FUNCTION "LGF_MatrixSubtraction" : Void
TITLE = LGF_MatrixSubtraction
{ S7_Optimized_Access := 'TRUE' }
AUTHOR : Siemens_Digital_Industries
FAMILY : LGF
NAME : LGF_MatrixSubtraction
//This function subtracts a matrix of the data type `ARRAY[*,*] of LREAL` from another one.
//
//The individual fields of the two matrices are read, subtracted and then output in the matrix `matrixResult`.
//
//$$
// result =
//
//\begin{bmatrix}
//   a_{11} & \cdots & a_{1n} \\
//   \vdots & \ddots & \vdots \\
//   a_{m1} & \cdots & a_{mn}
//\end{bmatrix}
//
//-
//
//\begin{bmatrix}
//   b_{11} & \cdots & b_{1n} \\
//   \vdots & \ddots & \vdots \\
//   b_{m1} & \cdots & b_{mn}
//\end{bmatrix}
//
//=
//
//\begin{bmatrix}
//   a_{11}-b_{11} & \cdots & a_{1n}-b_{1n} \\
//   \vdots & \ddots & \vdots \\
//   a_{m1}-b_{m1} & \cdots & a_{mn}-b_{mn}
//\end{bmatrix}
//$$
//
//Note
//:    Note that all input and output matrices must have the same number of columns and rows.
//
   VAR_OUTPUT
      error : Bool;   // FALSE: No error  TRUE: An error occurred during the execution of the FB
      status : Word;   // 16#0000-16#7FFF: Status of the FB  16#8000-16#FFFF: Error identification (see following Table)
   END_VAR

   VAR_IN_OUT
      matrix1 : Array[*, *] of LReal;   // First matrix - minuend
      matrix2 : Array[*, *] of LReal;   // Second matrix - subtrahend
      matrixResult : Array[*, *] of LReal;   // Sum of the matrices
   END_VAR

   VAR_TEMP
      tempMatrix1LowerBoundRows : DInt;   // Matrix1 lower bound for the rows (Dimension 1)
      tempMatrix1LowerBoundColumns : DInt;   // Matrix1 lower bound for the columns (Dimension 2)
      tempMatrix1UpperBoundRows : DInt;   // Matrix1 upper bound for the rows (Dimension 1)
      tempMatrix1UpperBoundColumns : DInt;   // Matrix1 upper bound for the columns (Dimension 2)
      tempMatrix2LowerBoundRows : DInt;   // Matrix2 lower bound for the rows (Dimension 1)
      tempMatrix2LowerBoundColumns : DInt;   // Matrix2 lower bound for the columns (Dimension 2)
      tempMatrix2UpperBoundRows : DInt;   // Matrix2 upper bound for the rows (Dimension 1)
      tempMatrix2UpperBoundColumns : DInt;   // Matrix2 upper bound for the columns (Dimension 2)
      tempResultMatrixLowerBoundRows : DInt;   // Result matrix lower bound for the rows (Dimension 1)
      tempResultMatrixLowerBoundColumns : DInt;   // Result matrix lower bound for the columns (Dimension 2)
      tempResultMatrixUpperBoundRows : DInt;   // Result matrix upper bound for the rows (Dimension 1)
      tempResultMatrixUpperBoundColumns : DInt;   // Result matrix upper bound for the columns (Dimension 2)
      tempCounterRows : DInt;   // Index counter for traversiong trough rows (Dimension 1)
      tempCounterColumns : DInt;   // Index counter for traversiong trough columns (Dimension 2)
   END_VAR

   VAR CONSTANT
      ROWS : UInt := 1;   // Rows are the first dimention of the two dimentional array
      COLUMNS : UInt := 2;   // Columns are the second dimension of the two dimensional array
      STATUS_NO_ERROR : Word := 16#0000;   // Execution finished without errors
      ERR_MATR1_LOWBOUND_ROWS_MATR2_LOWBOUND_ROWS : Word := 16#8200;   // Error: Matrix1 lower bound rows(Dim1) size is different with Matrix2 lower bound rows(Dim1)
      ERR_MATR1_LOWBOUND_ROWS_RESMATR_LOWBOUND_ROWS : Word := 16#8201;   // Error: Matrix1 lower bound rows(Dim1) size is different with Result Matrix lower bound rows(Dim1)
      ERR_MATR1_LOWBOUND_COLUMNS_MATR2_LOWBOUND_COLUMNS : Word := 16#8202;   // Error: Matrix1 lower bound columns(Dim2) size is different with Matrix 2 lower bound columns(Dim2)
      ERR_MATR1_LOWBOUND_COLUMNS_RESMATR_LOWBOUND_COLUMNS : Word := 16#8203;   // Error: Matrix1 lower bound columns(Dim2) size is different with Result Matrix lower bound columns(Dim2)
      ERR_MATR1_UPPBOUND_ROWS_MATR2_UPPBOUND_ROWS : Word := 16#8204;   // Error: Matrix1 upper bound rows(Dim1) size is different with Matrix2 upper bound rows(Dim1)
      ERR_MATR1_UPPBOUND_ROWS_RESMATR_UPPBOUND_ROWS : Word := 16#8205;   // Error: Matrix1 upper bound rows(Dim1)s size is different with Result Matrix upper bound rows(Dim1)
      ERR_MATR1_UPPBOUND_COLUMNS_MATR2_UPPBOUND_COLUMNS : Word := 16#8206;   // Error: Matrix1 upper bound columns(Dim2) size is different with Matrix2 upper bound columns(Dim2)
      ERR_MATR1_UPPBOUND_COLUMNS_RESMATR_UPPBOUND_COLUMNS : Word := 16#8207;   // Error: Matrix1 upper bound columns(Dim2) size is different with Result Matrix upper bound columns(Dim2)
   END_VAR


BEGIN
	REGION Block info header
	  //=============================================================================
	  // SIEMENS AG / (c)Copyright 2017
	  //-------------------------------------------------------------------------------
	  // Title:            LGF_MatrixSubtraction
	  // Comment/Function: Caluclates the difference of two matrices with same boundries
	  // Library/Family:   LGF(Library General Functions)
	  // Author:           Siemens Digital Industry Support
	  // Tested with:      S7-PLCSIM Advanced V2.0 SP1
	  // Engineering:      TIA Portal V15 Update 2
	  // Restrictions:     ENO disabled - error handling done by error and status
	  // Requirements:     PLC (S7-1200 / S7-1500)
	  //-------------------------------------------------------------------------------
	  // Change log table:
	  // Version  | Date       | Expert in charge       | Changes applied
	  //----------|------------|------------------------|------------------------------
	  // 01.00.00 19.08.2015  Siemens Industry Online Support
	  //                      First released version
	  // 01.00.01 02.01.2017  Siemens Industry Online Support
	  //                      Upgrade: TIA Portal V14 Update 1
	  // 02.00.00 06.02.2017  Siemens Industry Online Support
	  //                      Functionality using Array[*,*]
	  // 02.00.01 17.08.2018  Siemens Industry Online Support
	  //                      Upgrade: TIA V15 Update 2
	  // 02.00.06 07.10.2019  Simatic Systems Support
	  //                      Regions, comments and constants are added
	  //                      Moved matrices to IO field.
	  // 03.00.00 23.04.2020  Simatic Systems Support
	  //                      Set version to V3.0.0, harmonize the version of the whole library
	  // 03.00.01 02.02.2020  Simatic Systems Support
	  //                      Insert documentation
	  //=============================================================================
	END_REGION Block info header

	REGION Getting matrices size
	  //Determine the size of the matrices
	  // Lower bound rows
	  #tempMatrix1LowerBoundRows := LOWER_BOUND(ARR := #matrix1, DIM := #ROWS);
	  #tempMatrix2LowerBoundRows := LOWER_BOUND(ARR := #matrix2, DIM := #ROWS);
	  #tempResultMatrixLowerBoundRows := LOWER_BOUND(ARR := #matrixResult, DIM := #ROWS);
	  // Lower bound columns
	  #tempMatrix1LowerBoundColumns := LOWER_BOUND(ARR := #matrix1, DIM := #COLUMNS);
	  #tempMatrix2LowerBoundColumns := LOWER_BOUND(ARR := #matrix2, DIM := #COLUMNS);
	  #tempResultMatrixLowerBoundColumns := LOWER_BOUND(ARR := #matrixResult, DIM := #COLUMNS);

	  // Upper bound rows
	  #tempMatrix1UpperBoundRows := UPPER_BOUND(ARR := #matrix1, DIM := #ROWS);
	  #tempMatrix2UpperBoundRows := UPPER_BOUND(ARR := #matrix2, DIM := #ROWS);
	  #tempResultMatrixUpperBoundRows := UPPER_BOUND(ARR := #matrixResult, DIM := #ROWS);
	  // Upper bound columns
	  #tempMatrix1UpperBoundColumns := UPPER_BOUND(ARR := #matrix1, DIM := #COLUMNS);
	  #tempMatrix2UpperBoundColumns := UPPER_BOUND(ARR := #matrix2, DIM := #COLUMNS);
	  #tempResultMatrixUpperBoundColumns := UPPER_BOUND(ARR := #matrixResult, DIM := #COLUMNS);
	END_REGION

	REGION Error evaluation of matrixes dimentions
	  // Check the lower bound of all matrices
	  IF #tempMatrix1LowerBoundRows <> #tempMatrix2LowerBoundRows THEN
	    #error := TRUE;
	    #status := #ERR_MATR1_LOWBOUND_ROWS_MATR2_LOWBOUND_ROWS;
	    RETURN;
	  ELSIF #tempMatrix1LowerBoundRows <> #tempResultMatrixLowerBoundRows THEN
	    #error := TRUE;
	    #status := #ERR_MATR1_LOWBOUND_ROWS_RESMATR_LOWBOUND_ROWS;
	    RETURN;
	  ELSIF #tempMatrix1LowerBoundColumns <> #tempMatrix2LowerBoundColumns THEN
	    #error := TRUE;
	    #status := #ERR_MATR1_LOWBOUND_COLUMNS_MATR2_LOWBOUND_COLUMNS;
	    RETURN;
	  ELSIF #tempMatrix1LowerBoundColumns <> #tempResultMatrixLowerBoundColumns THEN
	    #error := TRUE;
	    #status := #ERR_MATR1_LOWBOUND_COLUMNS_RESMATR_LOWBOUND_COLUMNS;
	    RETURN;
	  END_IF;

	  // Check the upper bound of all matrices
	  IF (#tempMatrix1UpperBoundRows <> #tempMatrix2UpperBoundRows) THEN
	    #error := TRUE;
	    #status := #ERR_MATR1_UPPBOUND_ROWS_MATR2_UPPBOUND_ROWS;
	    RETURN;
	  ELSIF (#tempMatrix1UpperBoundRows <> #tempResultMatrixUpperBoundRows) THEN
	    #error := TRUE;
	    #status := #ERR_MATR1_UPPBOUND_ROWS_RESMATR_UPPBOUND_ROWS;
	    RETURN;
	  ELSIF (#tempMatrix1UpperBoundColumns <> #tempMatrix2UpperBoundColumns) THEN
	    #error := TRUE;
	    #status := #ERR_MATR1_UPPBOUND_COLUMNS_MATR2_UPPBOUND_COLUMNS;
	    RETURN;
	  ELSIF (#tempMatrix1UpperBoundColumns <> #tempResultMatrixUpperBoundColumns) THEN
	    #error := TRUE;
	    #status := #ERR_MATR1_UPPBOUND_COLUMNS_RESMATR_UPPBOUND_COLUMNS;
	    RETURN;
	  END_IF;
	END_REGION

	REGION Subtraction of the matrices and writting to output
	  FOR #tempCounterRows := #tempMatrix1LowerBoundRows TO #tempMatrix1UpperBoundRows DO
	    FOR #tempCounterColumns := #tempMatrix1LowerBoundColumns TO #tempMatrix1UpperBoundColumns DO
	      #matrixResult[#tempCounterRows, #tempCounterColumns] := #matrix1[#tempCounterRows, #tempCounterColumns] - #matrix2[#tempCounterRows, #tempCounterColumns];
	    END_FOR;
	  END_FOR;

	  #error := false;
	  #status := #STATUS_NO_ERROR;
	  // ENO mechanism is not used
	  ENO := TRUE;
	END_REGION

END_FUNCTION

